PROGRAM PRG_Machine
VAR
	

	
	//Forced Home
	Forced_Home_State						:INT:=0;
	Forced_Home_State_Next					:INT:=0;
	Forced_Home_Executed					:BOOL:=FALSE;

	//RepetitionCounter: INT;
	
	Pusher :FB_Pusher;
	Compress: FB_Compress;
	Shield: FB_Shield;

	ZenonStart: NT_StartProcess;
	//nameString: STRING;
	
	debug: INT;
	tickcounter: INT;
	tickcounter2: INT;

	State: INT:= 0;
	state_old: INT:=0;
	StateNext: INT:= 0;
	
	SM_StepRequest: BOOL:=FALSE;
	singleStep: BOOL:=FALSE;
		
	Clamp_Security_Time: TIME := T#30S;
	ClampTimer: TON;
	//DwellTimer: TON;
	//SaveTickCounter: INT := 0;

	DatumTaught: BOOL;
	//test: BOOL;
	//ReTeachOffsets: BOOL;
	//StopRequest: BOOL;
	//random: STRING(INT#4);
	rec_temp1: recipe;
	rec_temp2: recipe;
	rec_temp3: recipe;
	
END_VAR

IF TRUE THEN
	debug := debug+1;
END_IF



qbCompressServoTorqueLimit := 1000;
qbPusherServoTorqueLimit := 1000;
qbShieldServoTorqueLimit := 1000;


//The state-machine
CASE State OF
	
0: //Copy config .txt file into machine settings
	


	//Zenon start process function call - appears to never generate errors
	
	//IF ZenonStart.Busy=FALSE THEN
	ZenonStart (
		NETID :=,
		//PATHSTR := 'Hard Disk\CP6606_Runtime\zenonRCE.exe', //'C:\PROGRAM Files\COPA-DATA\zenon 7.20 SP0\Zenrt32.exe',
		//DIRNAME := 'Hard Disk\CP6606_Runtime',  //'C:\Program Files\COPA-DATA\zenon 7.20 SP0',
		PATHSTR := 'Hard Disk\ZenonRunTime\zenonRCE.exe', //'C:\PROGRAM Files\COPA-DATA\zenon 7.20 SP0\Zenrt32.exe',
		DIRNAME := 'Hard Disk\ZenonRunTime',  //'C:\Program Files\COPA-DATA\zenon 7.20 SP0',
		COMNDLINE := '',
		START := TRUE,
		TMOUT := DEFAULT_ADS_TIMEOUT
		);
	StateNext := 10;
	//END_IF	
	
	//IF ZenonStart.BUSY = FALSE THEN
	//	ZenonStart ( START := FALSE );
	//	StateNext := 10;
	//END_IF

10: //When restarting state machine, ensure E-Stop relay is not set
	//PRG_System.fbRecipeHandler.M_Next();
	qxEnableE_Stop := FALSE;
	tickcounter := 0;
	StateNext := 15;
	//qxEnableE_Stop:=TRUE;
15: //Check E-Stop relay is not set then Enable and initialise stuff - disable drive to clear errors
	//u are here
	
	//Shield._Reset();
	//Compress._Reset();
	//Pusher._Reset();
	

	//StartLoad := FALSE;
	ResetLampController.State := off;
	//RepetitionCounter := 0;
	//qxEnableE_Stop := TRUE;
	IF ixCabinetE_StopButtonOkay (*AND ixGuardRelayOkay*) THEN
		qxEnableE_Stop := TRUE;
		StateNext := 20;
	END_IF	
	
20: // Look for E-Stop button reset
	IF ixCabinetE_StopButtonOkay THEN
		ResetLampController.State := steady;
		sSystemStateMed := F_DisplayText("Press RESET button",0);	
		StateNext := 30;
	ELSE
		IF ixCabinetE_StopButtonOkay AND ixMachineE_StopButtonOkay THEN 
			ResetLampController.State := FastFlash;
			sSystemStateMed := F_DisplayText("Guard Open",0);
		ELSE
			ResetLampController.State := off;
			sSystemStateMed := F_DisplayText("E-Stop Depressed",0);
		END_IF
		CurrentProcessState	:= F_DisplayText("not ready",0);	//Main Screen	
	END_IF

30: // Wait for operator to hit reset button
	
	IF ixE_StopRelayOkay THEN
		ResetLampController.State := off;
		StateNext := 40;
		tickcounter := 0;
	ELSE
		tickcounter := tickcounter + 1;
		IF tickcounter >= 9800 THEN
			ResetLampController.State := steady;
			tickcounter := 0;
		END_IF
	END_IF

40: // look for guard closed - disable drive to clear errors
	sSystemStateMed := F_DisplayText("Guard Open",0);	
	CurrentProcessState	:= F_DisplayText("not ready",0);	//Main Screen	

	
	IF NOT ixGuardRelayOkay THEN
		ResetLampController.State := FastFlash;		
	ELSE
		ResetLampController.State := off;
		sSystemStateMed := F_DisplayText("Initialising Axes",0);	
		tickcounter := 0;
		StateNext := 100;
	END_IF
	
100: // wait 2 scans for power supply to drive to stabilise
	tickcounter := tickcounter + 1;
	IF tickcounter >= 2 THEN
		tickcounter := 0;
		StateNext := 110;
	END_IF

110: // prepare for Servo motion - enable drive
//you are here!!!!!!!!!!!!!!!!!!!!!!!!!!!!
	IF NOT ixResetButton THEN
		
		
	
		Shield._Enable();
		Pusher._Enable();
		Compress._Enable();
		
		tickcounter := tickcounter + 1;
		IF tickcounter >= 100 THEN
			tickcounter := 0;

			StateNext := 115;
		END_IF	
	END_IF


	
115: 
	
	//IF Shield.HomeExecuted = FALSE OR Pusher.HomeExecuted = FALSE OR Compress.HomeExecuted = FALSE THEN
	Stage_Name := 'Beginning';
	Maintenance_Visibility:=TRUE;
	qxStartButtonLamp:=TRUE;
	IF (ixStartButton OR Step_Next OR ixStart_Button_Machine) THEN
		IF (parameter_violation = FALSE) THEN
			qxStartButtonLamp:=FALSE;
			StateNext := 119;
			Step_Next := FALSE;
			Clamp_Alarm:=FALSE;
			Maintenance_Visibility:=FALSE;
			Stage_Name := 'Homing and Offsetting';

			rec_temp1:=Shield.Shield_Param;     
			rec_temp2:=Pusher.Pusher_Param;
			rec_temp3:=Compress.Compress_Param; 
		ELSE
			Step_Next:=FALSE;
		END_IF
	END_IF

	
119:
	IF rec_temp1.other.Shield_Home_Offset <> recipe_screen.Other.Shield_Home_Offset THEN
		Shield.HomeExecuted:=FALSE;
		Shield.OffsetExecuted:=FALSE;
	END_IF
	
	IF rec_temp2.other.Pusher_Home_Offset <> recipe_screen.Other.Pusher_Home_Offset THEN
		Pusher.HomeExecuted:=FALSE;
		Pusher.OffsetExecuted:=FALSE;
	END_IF
	
	IF rec_temp3.other.Compress_Home_Offset <> recipe_screen.Other.Compress_Home_Offset THEN
		Compress.HomeExecuted:=FALSE;
		Compress.OffsetExecuted:=FALSE;
	END_IF
	
	Shield.Shield_param:=recipe_screen;
	Compress.Compress_Param := recipe_screen;
	Pusher.Pusher_Param := recipe_screen;
	
	

	IF	Compress.HomeExecuted=FALSE OR Shield.HomeExecuted = FALSE OR Pusher.HomeExecuted = FALSE THEN
		statenext:=120;
	ELSE
		StateNext:=129;
	END_IF
		
120: //you are here!!!!!!!!!!!!

	
	
	IF Pusher.HomeExecuted = FALSE THEN 
		Pusher._Home();
	END_IF
	
	IF Compress.HomeExecuted = FALSE THEN
		Compress._Home();
	END_IF
	
	
	IF Compress.HomeExecuted AND Pusher.HomeExecuted THEN
		StateNext := 125;                //directly to end
		//Compress.HomeExecuted:=FALSE;
		//Pusher.HomeExecuted:=FALSE;
		
	END_IF
	
125:
	//random:='arda';
	IF Shield.HomeExecuted = FALSE THEN
		Shield._Home();
		
	ELSE
		StateNext := 128;
		//Shield.HomeExecuted := FALSE;
	END_IF
128:
		

	IF Compress.OffsetExecuted = FALSE THEN
		Compress.Offset();
	END_IF
	
	IF Shield.OffsetExecuted = FALSE THEN
		Shield.Offset();
	END_IF
	
	IF Pusher.OffsetExecuted = FALSE THEN
		Pusher.Offset();
	END_IF
	
	IF Pusher.OffsetExecuted AND Shield.OffsetExecuted AND Compress.OffsetExecuted THEN
		Maintenance_Visibility := TRUE;
		qxStartButtonLamp:=TRUE;
		IF (ixStartButton OR Step_Next OR ixStart_Button_Machine) THEN
			IF (parameter_violation =FALSE) THEN
				qxStartButtonLamp:=FALSE;
				Shield.Shield_param:=recipe_screen;
				Compress.Compress_Param := recipe_screen;
				Pusher.Pusher_Param := recipe_screen;
			
				StateNext:=130;
				Step_Next:=FALSE;
				Maintenance_Visibility := FALSE;
			ELSE
				Step_Next:=FALSE;
			END_IF
		END_IF
	END_IF
	
	

129: //debug	
	
	IF Debug_Mode THEN
		Maintenance_Visibility := TRUE;
		IF Step_Next THEN
			IF Parameter_Violation = FALSE THEN
				Step_Next:=FALSE;
				StateNext:=130;
				Maintenance_Visibility := FALSE;
			
				Shield.Shield_param:=recipe_screen;
				Compress.Compress_Param := recipe_screen;
				Pusher.Pusher_Param := recipe_screen;
			ELSE
				Step_Next:=FALSE;
			END_IF
		END_IF
	ELSE
		StateNext:=130;
		Maintenance_Visibility := FALSE;
	END_IF
		
130: //stage 1
	Stage_Name := 'Compress Tobacco';
	IF qxClamp = FALSE THEN
		qxClamp:=TRUE;
		ClampTimer.IN:=TRUE;
		ClampTimer.PT:=Clamp_Security_Time;

	END_IF
	
	IF Compress.Stage1Executed = FALSE THEN
		IF state_old = 130 THEN
			Message:='I am trying to continue';
		END_IF 
		Compress._Stage1();
		Compress.HomeExecuted:=FALSE;	
	ELSE
		//Compress.Stage1Executed := FALSE;
		StateNext := 131;
		DatumTaught := FALSE;
	END_IF

131: //debug

	IF Debug_Mode THEN
		Maintenance_Visibility := TRUE;
		IF Step_Next THEN
			IF Parameter_Violation = FALSE THEN
				Step_Next:=FALSE;
				StateNext:=135;
				Maintenance_Visibility := FALSE;
			
				Shield.Shield_param:=recipe_screen;
				Compress.Compress_Param := recipe_screen;
				Pusher.Pusher_Param := recipe_screen;
			ELSE
				Step_Next:=FALSE;
			END_IF
		END_IF
	ELSE
		StateNext:=135;
		Maintenance_Visibility := FALSE;
	END_IF
	
135://stage2
	Stage_Name := 'Load Tobacco';
	Compress.Stage1Executed := FALSE;
	
	IF Pusher.Stage2Executed = FALSE THEN
		Pusher._Stage2();
		Pusher.HomeExecuted:=FALSE;
	END_IF
	
	IF Shield.Stage2Executed = FALSE THEN
		Shield._Stage2();
		Shield.HomeExecuted:=FALSE;
	END_IF
	
	IF Shield.Stage2Executed AND Pusher.Stage2Executed THEN
		//Shield.Stage2Executed:=FALSE;
		//Pusher.Stage2Executed:=FALSE;
		//DatumTaught:=FALSE;
		StateNext := 137;
	END_IF
137: //debug

	IF Debug_Mode THEN
		Maintenance_Visibility := TRUE;
		IF Step_Next THEN
			IF Parameter_Violation = FALSE THEN
				Step_Next:=FALSE;
				StateNext:=140;
				Maintenance_Visibility := FALSE;
			
				Shield.Shield_param:=recipe_screen;
				Compress.Compress_Param := recipe_screen;
				Pusher.Pusher_Param := recipe_screen;
			ELSE
				Step_Next:=FALSE;
			END_IF
		END_IF
	ELSE
		StateNext:=140;
		Maintenance_Visibility := FALSE;
	END_IF
	
140: //stage3
	
	Stage_Name := 'Shield Retract';
	
	Shield.Stage2Executed:=FALSE;
	Pusher.Stage2Executed:=FALSE;
	
	IF	Shield.Stage3Executed = FALSE THEN
		Shield._Stage3();
		Shield.HomeExecuted:=FALSE;	
	ELSE
		//Shield.Stage3Executed := FALSE;
		StateNext := 141;
		DatumTaught := FALSE;
	END_IF

141: //debug

	IF Debug_Mode THEN
		Maintenance_Visibility := TRUE;
		IF Step_Next THEN
			IF Parameter_Violation = FALSE THEN
				Step_Next:=FALSE;
				StateNext:=142;
				Maintenance_Visibility := FALSE;
			
				Shield.Shield_param:=recipe_screen;
				Compress.Compress_Param := recipe_screen;
				Pusher.Pusher_Param := recipe_screen;
			ELSE
				Step_Next:=FALSE;
			END_IF
		END_IF
	ELSE
		StateNext:=142;
		Maintenance_Visibility := FALSE;
	END_IF	
	
142: //Tamp
	
	Stage_Name := 'Tamp';
	
	Shield.Stage3Executed := FALSE;
	
	IF	Pusher.TampExecuted = FALSE THEN
		Pusher.Tamp();
		Pusher.HomeExecuted:=FALSE;	
	ELSE
		StateNext := 143;
	END_IF
	
143: //debug

	IF Debug_Mode THEN
		Maintenance_Visibility := TRUE;
		IF Step_Next THEN
			IF Parameter_Violation = FALSE THEN
				Step_Next:=FALSE;
				StateNext:=145;
				Maintenance_Visibility := FALSE;
			
				Shield.Shield_param:=recipe_screen;
				Compress.Compress_Param := recipe_screen;
				Pusher.Pusher_Param := recipe_screen;
			ELSE
				Step_Next:=FALSE;
			END_IF
		END_IF
	ELSE
		StateNext:=145;
		Maintenance_Visibility := FALSE;
	END_IF
	
145: //stage4
	
	Stage_Name := 'Eject Spill';
	
	Pusher.TampExecuted := FALSE;
	IF	Pusher.Stage4Executed = FALSE THEN
		Pusher._Stage4();
		Pusher.HomeExecuted:=FALSE;	
	ELSE
		//Pusher.Stage4Executed := FALSE;
		StateNext := 147;
		DatumTaught := FALSE;
	END_IF

147: //debug

	IF Debug_Mode THEN
		Maintenance_Visibility := TRUE;
		IF Step_Next THEN
			IF Parameter_Violation = FALSE THEN
				Step_Next:=FALSE;
				StateNext:=150;
				Maintenance_Visibility := FALSE;
			
				Shield.Shield_param:=recipe_screen;
				Compress.Compress_Param := recipe_screen;
				Pusher.Pusher_Param := recipe_screen;
			ELSE
				Step_Next:=FALSE;
			END_IF
		END_IF
	ELSE
		StateNext:=150;
		Maintenance_Visibility := FALSE;
	END_IF
	
150: //stage 5
	
	Stage_Name := 'Retract All';
	
	Pusher.Stage4Executed := FALSE;
	IF Pusher.Stage5Executed = FALSE THEN
		Pusher._Stage5();
		Pusher.HomeExecuted:=FALSE;
	END_IF
	
	IF Compress.Stage5Executed = FALSE THEN
		Compress._Stage5();
		Compress.HomeExecuted:=FALSE;
	END_IF
	
	IF Compress.Stage5Executed AND Pusher.Stage5Executed THEN
		//Compress.Stage5Executed:=FALSE;
		//Pusher.Stage5Executed:=FALSE;
		DatumTaught:=FALSE;
		StateNext := 155;
	END_IF	
151:
	Pusher._Halt();
	Shield._Halt();
	Compress._Halt();
	IF Pusher.PusherServo.xhalted AND Shield.ShieldServo.xHalted AND Compress.CompressServo.xHalted AND (ixStartbutton OR ixStart_Button_Machine) THEN
		Pusher._Halt_false();
		Shield._Halt_false();
		Compress._Halt_false();
		Pusher._Soft_Reset();
		Shield._Soft_Reset();
		Compress._Soft_Reset();
		statenext:=state_old;
	END_IF

155: //end
	Compress.Stage5Executed:=FALSE;
	Pusher.Stage5Executed:=FALSE;
	
	Pusher.HomeExecuted:= TRUE;
	Shield.HomeExecuted:=TRUE;
	Compress.HomeExecuted:=TRUE;
	statenext:= 115;

	
1000: // overtorque
	CurrentProcessState	:= F_DisplayText("Process incomplete",0);			//Main Screen
	//StartLoad := FALSE;
	
	Compress._Reset();
	Pusher._Reset();
	Shield._Reset();
	
	qxclamp:=FALSE;
	ClampTimer.IN:=FALSE;
	ClampTimer.PT:=Clamp_Security_Time;
	
	statenext:=2000;
	
	
	

	
2000: // guard and estop
	
	tickcounter:= tickcounter+1;
	IF	tickcounter = 100 THEN
		tickcounter:=0;
		statenext:=15;
		overtorque_alarm:=FALSE;
	END_IF

2010: // clamp alarm
	
	tickcounter:= tickcounter+1;

	
	IF clamp_alarm THEN
		
		IF	tickcounter = 3000 THEN
			tickcounter:=0;
			statenext:=100;
			Clamp_Cooling := FALSE;
			Clamp_Alarm := FALSE;
		ELSE
			Clamp_Cooling := TRUE;
			
			IF Pusher.PusherServo.xstopped AND Shield.ShieldServo.xstopped AND Compress.CompressServo.xstopped THEN
				Pusher._Reset();
				Shield._Reset();
				Compress._Reset();
			END_IF
		END_IF
	ELSE
		IF	tickcounter = 100 THEN
			tickcounter:=0;
			statenext:=100;
			Clamp_Cooling := FALSE;
		ELSIF Pusher.PusherServo.xstopped AND Shield.ShieldServo.xstopped AND Compress.CompressServo.xstopped THEN
			Pusher._Reset();
			Shield._Reset();
			Compress._Reset();
			
		END_IF
	END_IF
	
2020: //force home
(*	
	IF Forced_Home_Executed = FALSE THEN
		Handle_Forced_Home();	
	ELSE
		StateNext:=115;
		Forced_Home_Executed:=FALSE;
	END_IF
*)
	
END_CASE

Pusher._Update();
Shield._Update();
Compress._Update();
ClampTimer();

IF 	StateNext <> 115 AND 
	StateNext <> 128 THEN
	qxStartButtonLamp:=FALSE;
END_IF

IF 	StateNext <> 115 AND 
	StateNext <> 128 AND 
	StateNext <> 129 AND 
	StateNext <> 131 AND 
	StateNext <> 137 AND 
	StateNext <> 141 AND 
	StateNext <> 143 AND 
	StateNext <> 147 THEN

	Maintenance_Visibility := FALSE;
END_IF

//Motor Overtorque
IF StateNext >= 110 AND StateNext <= 155  THEN					// machine is running
	
	IF ibCompressServoTorque  > 2000 OR ibCompressServoTorque  < -2000 THEN						// PuckSlideServo torque too high
		//Message := WSTRING_TO_STRING("Tobacco Compress Servo over-torque");
		StateNext := 1000;
		tickcounter:=0;
		overtorque_alarm:= TRUE;	
	END_IF
	
	IF ibPusherServoTorque  > 2000 OR ibPusherServoTorque  < -2000 THEN						// HeaterSlideServo torque too high
		//Message := WSTRING_TO_STRING("Rod Pusher Servo over-torque");
		StateNext := 1000;
		tickcounter:=0;
		overtorque_alarm:= TRUE;	
	END_IF
	
	IF ibShieldServoTorque  > 2000 OR ibShieldServoTorque  < -2000 THEN						// HeaterSlideServo torque too high
		//Message := WSTRING_TO_STRING("Rod Shield Servo over-torque");
		StateNext := 1000;
		tickcounter:=0;
		overtorque_alarm:= TRUE;	
	END_IF
END_IF


//Toggole Clamp
IF (StateNext >= 115 AND StateNext <= 155) AND Toggle_Clamp THEN
	Toggle_Clamp := FALSE;
	IF qxClamp = FALSE THEN
		
		qxClamp:=TRUE;
		ClampTimer.IN:=TRUE;
		ClampTimer.PT:=Clamp_Security_Time;

	ELSE
		
		qxClamp:=FALSE;
		ClampTimer.IN:=FALSE;
		ClampTimer.PT:=Clamp_Security_Time;
		
	END_IF
	
	
END_IF

//stop button
IF NOT ixstop_button AND (Statenext<>151) THEN
	//	state_old:=statenext;
	//	statenext:= 151;
	tickcounter:=0;
	//Message:='Clamp Overtime';
	qxClamp:=FALSE;

	
	ClampTimer.IN:=FALSE;
	ClampTimer.PT:=Clamp_Security_Time;
	
	
	
	Compress._mc_stop();
	Shield._mc_stop();
	Pusher._mc_stop();
	StateNext := 2010;
	
	
END_IF

//Clamp Err
IF (Clamptimer.Q=TRUE) AND StateNext >= 100 AND StateNext <= 155 THEN 
	
	tickcounter:=0;
	//Message:='Clamp Overtime';
	qxClamp:=FALSE;

	
	ClampTimer.IN:=FALSE;
	ClampTimer.PT:=Clamp_Security_Time;
	
	Clamp_Alarm:=TRUE;
	
	Compress._mc_stop();
	Shield._mc_stop();
	Pusher._mc_stop();
	StateNext := 2010;

END_IF

//Home
IF (Force_Home) AND StateNext >= 115 AND StateNext <= 155 THEN 
	Force_Home:=FALSE;
	StateNext := 2020;
	tickcounter:=0;
	
	
	
	qxclamp:=FALSE;
	ClampTimer.IN:=FALSE;
	ClampTimer.PT:=Clamp_Security_Time;
	
	Pusher._Reset();
	Shield._Reset();
	Compress._Reset();
END_IF

//guard
IF (NOT ixGuardRelayOkay) AND StateNext >= 100 AND StateNext <= 155 THEN 
	
	StateNext := 2000;
	tickcounter:=0;
	
	//Message:='Guard Open';
	
	qxclamp:=FALSE;
	ClampTimer.IN:=FALSE;
	ClampTimer.PT:=Clamp_Security_Time;
	
	IF Pusher.HomeExecuted= FALSE OR Shield.HomeExecuted = FALSE OR Compress.HomeExecuted = FALSE THEN
		Pusher._Reset();
		Shield._Reset();
		Compress._Reset();
	ELSE
		Pusher._Reset_Medium();
		Shield._Reset_Medium();
		Compress._Reset_Medium();
	END_IF
END_IF

//estop
IF (NOT ixCabinetE_StopButtonOkay) AND StateNext >= 30 AND StateNext <= 155 THEN 
	
	tickcounter:=0;
	
	//Message:='E-stop Pressed';
	
	qxclamp:=FALSE;
	ClampTimer.IN:=FALSE;
	ClampTimer.PT:=Clamp_Security_Time;
	

	
	//IF Compress.CompressServo.xStopped AND Shield.ShieldServo.xStopped AND Pusher.PusherServo.xStopped THEN
	StateNext := 2000;
	Pusher._Reset();
	Shield._Reset();
	Compress._Reset();
	//END_IF
END_IF

//IF State <> StateNext THEN - step through the state machine if required
IF singleStep AND statenext > 119 THEN
	//IF NOT SM_StepRequest THEN
	//	SM_StepRequest := TRUE; 
	//END_IF
	IF SM_StepRequest THEN
		SM_StepRequest := FALSE;
		State := StateNext;
	END_IF
ELSE
	State := StateNext;
END_IF

PROPERTY ext_Clamp_Security_Time : TIME
GET
ext_Clamp_Security_Time := Clamp_Security_Time;
END_GET
SET
Clamp_Security_Time := ext_Clamp_Security_Time;
END_SET
END_PROPERTY

PROPERTY ext_ClampTimer : TON
GET
ext_ClampTimer:=ClampTimer;
END_GET
SET
ClampTimer:=ext_ClampTimer;
END_SET
END_PROPERTY

METHOD Handle_Forced_Home
VAR_INPUT
END_VAR
CASE Forced_Home_State OF
	
0:	
	tickcounter:=tickcounter + 1;
	IF tickcounter = 100 THEN
		Forced_Home_State_Next:=5;
	END_IF
5:	



END_CASE

Forced_Home_State_Next := Forced_Home_State;
END_METHOD

METHOD StopClampTimer
VAR_INPUT
END_VAR
ClampTimer.IN:=FALSE;
ClampTimer.PT:= Clamp_Security_Time;
END_METHOD

END_PROGRAM

(* stored: Version 1.1.0.1, ProductVersion 3.1.4020.12
   POU PRG_Machine: Id {4059ff51-9b15-4d7b-8b65-432c3cf02eab}, SpecialFunc None
   Property ext_Clamp_Security_Time: Id {b4a0574a-c59c-4187-912c-e138bff48456}
   Get Get: Id {6f9cde7b-b8c0-4b49-bc66-95e4a3439a9f}
   Set Set: Id {8abc84f1-4a75-4404-9fee-f285ee2e4ef0}
   Property ext_ClampTimer: Id {14e072fb-8285-42c1-9c45-0d63393dfcd2}
   Get Get: Id {321e20e3-e34b-4a23-ae19-a8f738310bcc}
   Set Set: Id {f0e4832a-6e15-4cc1-ab7a-c4491ec3cf3f}
   Method Handle_Forced_Home: Id {04eb6cdf-a7b3-4b41-a49a-21ff121f07e9}
   Method StopClampTimer: Id {d74d2087-e1fa-4163-bf2f-94ebc8b0fc77} *)
